(* PLC project Unnamed, Unknown Unnamed 1 *)
(* stored: creationDateTime 2019-12-06T10:28:35, modificationDateTime 2019-12-11T12:37:34 *)

PROGRAM program1
  VAR
    temp_sensor AT %IW100 : INT;
    temperatura AT %MW101 : INT;
    analog_lamp AT %QW100 : UINT;
    led_alarm AT %QX100.0 : BOOL;
  END_VAR

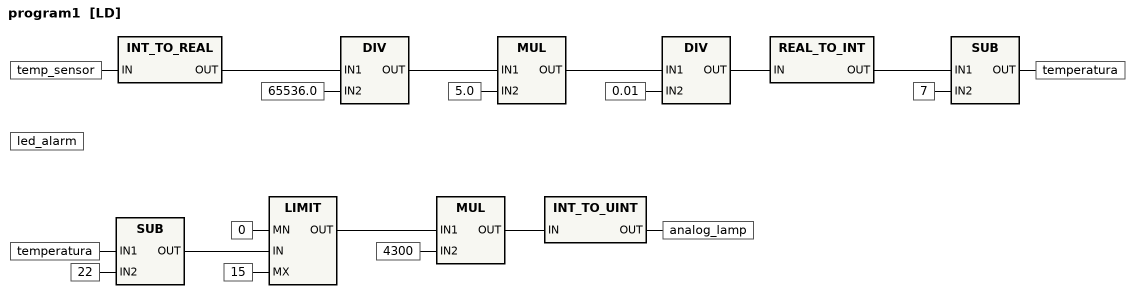
(* LD diagram, written out as Structured Text *)
analog_lamp := INT_TO_UINT(LIMIT(0, temperatura - 22, 15) * 4300);
temperatura := REAL_TO_INT(INT_TO_REAL(temp_sensor) / 65536.0 * 5.0 / 0.01) - 7;
(* drawn but not wired to any output: led_alarm *)
END_PROGRAM

CONFIGURATION Config0
  RESOURCE Res0 ON PLC
    TASK task0(INTERVAL := T#20ms, PRIORITY := 0);
    PROGRAM instance0 WITH task0 : program1;
  END_RESOURCE
END_CONFIGURATION
